Staubli VAL3: message.pgx

public program message(string& x_sMessage[], num x_nIndex)
begin
  // load the default one
  call language:message(x_sMessage,x_nIndex)
end
